(* PLC project undeclared, plcc plcc tests 1 *)
(* stored: creationDateTime 2026-09-27T00:00:00 *)

PROGRAM Undeclared
  VAR
    A : BOOL;
  END_VAR

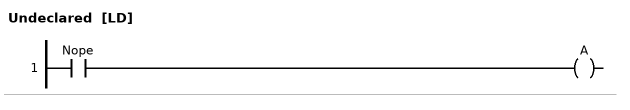
(* LD diagram, written out as Structured Text *)
A := Nope;
END_PROGRAM
